FUNCTION_BLOCK PedLightCtl_AT (* Function block for controling the operation of a pedestrian trafic light with one red and one green light *)
  (* Standard: 61499-2 *)
  (* Version 0.0, 2014-07-11, 4DIAC-IDE, 4DIAC-Consortium *)
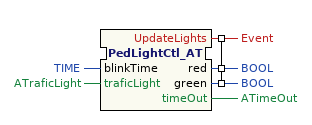
  EVENT_OUTPUT
    UpdateLights WITH green, red;
  END_EVENT
  VAR_INPUT
    blinkTime : TIME;
  END_VAR
  VAR_OUTPUT
    red : BOOL;
    green : BOOL;
  END_VAR
  SOCKETS
    traficLight : ATraficLight;
  END_SOCKETS
  PLUGS
    timeOut : ATimeOut;
  END_PLUGS
  VAR
    blinkCount : UINT; (* Internal Variable *)
  END_VAR
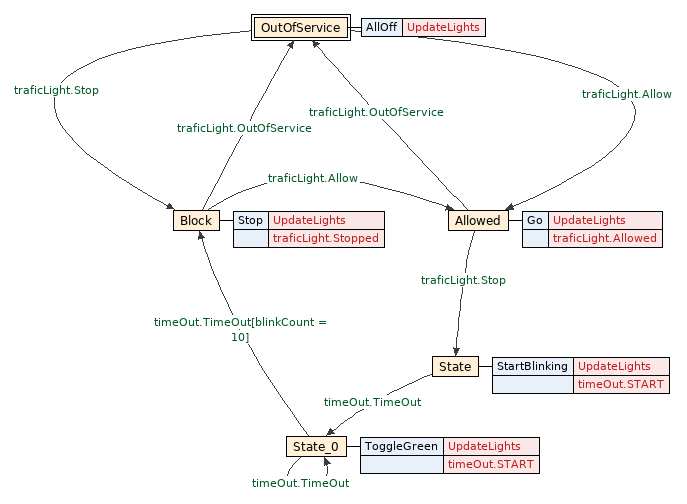
  EC_STATES
    OutOfService : AllOff -> UpdateLights;
    Block : Stop -> UpdateLights, -> traficLight.Stopped;
    Allowed : Go -> UpdateLights, -> traficLight.Allowed;
    State : StartBlinking -> UpdateLights, -> timeOut.START;
    State_0 : ToggleGreen -> UpdateLights, -> timeOut.START;
  END_STATES
  EC_TRANSITIONS
    OutOfService TO Block := traficLight.Stop;
    Block TO OutOfService := traficLight.OutOfService;
    Block TO Allowed := traficLight.Allow;
    Allowed TO OutOfService := traficLight.OutOfService;
    OutOfService TO Allowed := traficLight.Allow;
    Allowed TO State := traficLight.Stop;
    State TO State_0 := timeOut.TimeOut;
    State_0 TO Block := timeOut.TimeOut[blinkCount = 10];
    State_0 TO State_0 := timeOut.TimeOut;
  END_TRANSITIONS
  ALGORITHM AllOff IN ST:
red := FALSE;
green := FALSE;
  END_ALGORITHM
  ALGORITHM Stop IN ST: (* Put lights in stop mode (i.e., red := true, green := false) *)
red := TRUE;
green := FALSE;
  END_ALGORITHM
  ALGORITHM Go IN ST: (* Put lights in Walk mode (i.e., red := false, green := true) *)
red := FALSE;
green := TRUE;
  END_ALGORITHM
  ALGORITHM StartBlinking IN ST: (* new algorithm *)
timeOut.DT := blinkTime;
blinkCount := 0;
green := FALSE;
  END_ALGORITHM
  ALGORITHM ToggleGreen IN ST: (* new algorithm *)
green := NOT green;
blinkCount := blinkCount + 1;
  END_ALGORITHM
END_FUNCTION_BLOCK
